// TIA Portal V18 export
FUNCTION "PIDSupplyTempHeating" : Void   // FC10, FBD
{ S7_Optimized_Access := 'TRUE' }
VERSION : 0.1
// stored: AutoNumber false, IsIECCheckEnabled false, SetENOAutomatically false, UDAEnableTagReadback false
   VAR_INPUT
      UnitID : Int;
      Actual : Real;
      SetPoint : Real;
   END_VAR
   VAR_OUTPUT
      PIDOutput : Real;
   END_VAR
BEGIN
END_FUNCTION
